// TIA Portal V16 export
// export: Created 2025-12-30T17:36:41.3348066Z, ExportSetting WithDefaults, DisplayName Totally Integrated Automation Portal, DisplayVersion V16, DisplayName TIA Portal Version Control Interface, DisplayVersion V16, DisplayName TIA Portal Openness, DisplayVersion V16, DisplayName STEP 7 Professional, DisplayVersion V16, DisplayName STEP 7 Safety, DisplayVersion V16, DisplayName WinCC Professional, DisplayVersion V16
DATA_BLOCK "FB_Assembler_Logic_DB"   // DB1
VERSION : 0.1
// stored: AutoNumber true, InstanceOfName FB_Assembler_Logic, InstanceOfType FB
"FB_Assembler_Logic"
   // VAR_INPUT
   //    "Moving X" : Bool;
   //    "Moving Z" : Bool;
   //    "Item detected" : Bool;
   //    "Lid at place" : Bool;
   //    "Lid clamped" : Bool;
   //    "Pos. at limit (lids)" : Bool;
   //    "Base at place" : Bool;
   //    "Base clamped" : Bool;
   //    "Pos. at limit (bases)" : Bool;
   //    "Part leaving" : Bool;
   //    Start : Bool;
   //    Reset : Bool;
   //    Stop : Bool;
   //    "Emergency stop" : Bool;
   //    Auto : Bool;
   //    "FACTORY I/O (Uruchomiony)" : Bool;
   //    "Reset Coutner" : Bool;
   // END_VAR
   // VAR_OUTPUT
   //    "Move X" : Bool;
   //    "Move Z" : Bool;
   //    Grab : Bool;
   //    "Lids conveyor" : Bool;
   //    "Clamp lid" : Bool;
   //    "Pos. raise (lids)" : Bool;
   //    "Bases conveyor" : Bool;
   //    "Clamp base" : Bool;
   //    "Pos. raise (bases)" : Bool;
   //    "Start light" : Bool;
   //    "Reset light" : Bool;
   //    "Stop light" : Bool;
   //    "Counter" : DInt;
   //    "Reset Coutner Light" : Bool;
   // END_VAR
   // VAR
   //    stat_Step : Int;
   //    stat_TrigLid : F_TRIG;
   //    stat_TrigBase { S7_SetPoint := 'True'} : F_TRIG;
   //    stat_LidDone { S7_SetPoint := 'True'} : Bool;
   //    stat_BaseDone : Bool;
   //    timerLift : TON_TIME;
   //    stat_HoldingPart { S7_SetPoint := 'True'} : Bool;
   //    stat_X_Started : Bool;
   //    stat_Z_Started : Bool;
   //    System_Pracuje : Bool;
   //    Awaria_Aktywna : Bool;
   // END_VAR
BEGIN
END_DATA_BLOCK
